// TIA Portal project "LavaCoches_IgnacioMorillasPadial_II" (V15)

(* hardware
DEVICE "S7300/ET200M station_1"  S7-300 station
   slot 0: "Perfil soporte_0"  Rail  6ES7 390-1***0-0AA0
   slot 2: "PLC_1"  CPU 314C-2 PN/DP  6ES7 314-6EH04-0AB0  V3.3
      slot 2: "Interfaz PROFINET_1"  PN-IO
         slot 1: "Port_1"  Port
         slot 2: "Port_2"  Port
      slot 5: "DI 24/DO 16_1"  DI24/DO16
      slot 6: "AI 5/AO 2_1"  AI5/AO2
      slot 7: "Contaje_1"  Counter
      slot 8: "Posicionamiento_1"  Positioning
*)

// ===== PLC "PLC_1"  CPU 314C-2 PN/DP =====

VAR_GLOBAL   // PLC tag table "STEP7 classic symbols"
   "CV2_FU" AT %I12.2 : Bool;   // Cepillo Vertical Izquierdo Fuera
   "CV2_Me" AT %I12.1 : Bool;   // Cepillo Vertical Izquierdo Medio
   "CV2_De" AT %I12.0 : Bool;   // Cepillo Vertical Izquierdo Dentro
   "V_Luz2" AT %I8.5 : Bool;   // Ventilador Sensor de Luz 2
   "V_Luz1" AT %I8.4 : Bool;   // Ventilador Sensor de Luz 1
   "CH_Abajo" AT %I8.3 : Bool;   // Cepillo Horizontal Sensor Magnético Abajo
   "CR2_Recoger" AT %Q9.3 : Bool;   // Cepillo Rueda Derecho Control Retirada
   "CR2_Salir" AT %Q9.2 : Bool;   // Ceplilo Rueda Derecho Control Salida
   "CR1_Recoger" AT %Q9.1 : Bool;   // Cepillo Rueda Izquierda Control Retirada
   "CV1_Fu" AT %I9.5 : Bool;   // Cepillo Vertical Derecho Fuera
   "CH_Bajar" AT %Q8.2 : Bool;   // Cepillo Horizontal Control Bajar
   "CRE_Avanzar" AT %Q8.1 : Bool;   // Cremallera Conrtol Avanzar
   "CRE_Retroceder" AT %Q8.0 : Bool;   // Cremallera Control Retroceder
   "CV2_R" AT %Q12.3 : Bool;   // Cepillo Vertical Derecho Rotar
   "CV1_De" AT %I9.7 : Bool;   // Cepillo Vertical Derecho Dentro
   "CV1_Me" AT %I9.6 : Bool;   // Cepillo Vertical Derecho Medio
   "CV2_Salir" AT %Q12.2 : Bool;   // Cepillo Vertical Izquierdo Salir
   "CR1_De" AT %I9.0 : Bool;   // Cepillo Rueda Derecha Dentro
   "V_Abajo" AT %I8.7 : Bool;   // Ventilador Sensor Magnético Abajo
   "V_Arriba" AT %I8.6 : Bool;   // Ventilador Sensor Magnético Arriba
   "Cont_CV" AT %MW10 : Int;   // Contador Ciclos CV
   "CV1_Salir" AT %Q12.1 : Bool;   // Cepillo Vertical Derecho Salir
   "CV1_R" AT %Q12.0 : Bool;   // Cepillo Vertical Derecho Rotar
   "CV1_Recoger" AT %Q9.7 : Bool;   // Cepillo Vertical Derecho Recoger
   "CH_Arriba" AT %I8.2 : Bool;   // Cepillo Horizontal Sensor Magnético Arriba
   "CH_Luz2" AT %I8.1 : Bool;   // Cepillo Horizontal Sensor de Luz 2
   "CH_Luz1" AT %I8.0 : Bool;   // Cepillo Horizontal Sensor de Luz 1
   "CR1_Salir" AT %Q9.0 : Bool;   // Cepillo Rueda Izquierda Control Salida
   "V_Subir" AT %Q8.7 : Bool;   // Ventilador Control Subir
   "CH_Subir" AT %Q8.6 : Bool;   // Cepillo Horizontal Control Subir
   "CV_Frente" AT %I12.7 : Bool;   // Cremallera Posción Labado Delante
   "CV_Atrás" AT %I12.6 : Bool;   // Cremallera Posción Labado Atrás
   "CR_Frente" AT %I12.5 : Bool;   // Cremallera Posición Ruedas Delanteras
   "CR2_Fu" AT %I9.2 : Bool;   // Cepillo Rueda Izquierda Fuera
   "CR2_De" AT %I9.3 : Bool;   // Cepillo Rueda Izquierda Dentro
   "CR1_Fu" AT %I9.1 : Bool;   // Cepillo Rueda Derecha Fuera
   "CH_R_+" AT %Q8.5 : Bool;   // Cepillo Horizontal Rotación Horaria
   "CH_R_-" AT %Q8.4 : Bool;   // Cepillo Horizontal Rotación Antihoraria
   "V_Bajar" AT %Q8.3 : Bool;   // Ventilador Control Bajar
   "CRE_Final" AT %I12.4 : Bool;   // Cremallera Posción Final
   "CRE_Inicio" AT %I12.3 : Bool;   // Cremallera Posición Inicio
   "CR_Atrás" AT %I13.0 : Bool;   // Cremallera Posción Ruedas Traseras
   "CV2_Recoger" AT %Q9.6 : Bool;   // Cepillo Vertical Izquierdo Recoger
   "CR2_R" AT %Q9.5 : Bool;   // Cepillo Izquierdo Rueda Rotación Horaria
   "CR1_R" AT %Q9.4 : Bool;   // Cepillo Derecho Rueda Rotación Horaria
   "CRE_Avanzar_CM" AT %M0.0 : Bool;
   "CRE_Retroceder_CM" AT %M0.2 : Bool;
   "CV1_Salir_CM" AT %M0.3 : Bool;
   "CV1_Recoger_CM" AT %M0.4 : Bool;
   "CV1_R_CM" AT %M0.5 : Bool;
   "CV2_Salir_CM" AT %M0.6 : Bool;
   "CV2_Recger_CM" AT %M0.7 : Bool;
   "CV2_R_CM" AT %M1.0 : Bool;
   "CH_Bajar_CM" AT %M1.1 : Bool;
   "CH_Subir_CM" AT %M1.2 : Bool;
   "CH_R_+_CM" AT %M1.3 : Bool;
   "CH_R_-_CM" AT %M1.4 : Bool;
   "V_Bajar_CM" AT %M1.5 : Bool;
   "V_Subir_CM" AT %M1.6 : Bool;
   "Reset_Maqueta" AT %M1.7 : Bool;
   "Automatico_Manual" AT %M0.1 : Bool;
   "AUX" AT %M2.0 : Bool;
   "AUX2" AT %M2.1 : Bool;
END_VAR

FUNCTION "Estructura horizontal" : Void   // FC1, SCL
{ S7_Optimized_Access := 'FALSE' }
VERSION : 0.1
BEGIN
   IF "CRE_Avanzar_CM" AND NOT "Automatico_Manual" THEN

       // sube hasta que ambos sensores opticos estan activos, o finalcarrera de arriba.
       IF "CH_Luz1" AND "CH_Luz2" THEN
           "CH_Subir_CM" := 0;
           "CH_Subir" := 0;
           "CH_Bajar_CM" := 1;
           "CH_Bajar" := 1;
       END_IF;

       // baja hasta que alguno de los sensores opticos mande una señal o llegue al final de carrera abajo.
       IF NOT "CH_Luz1" OR NOT "CH_Luz2" THEN
           "CH_Subir_CM" := 1;
           "CH_Subir" := 1;
       END_IF;
   END_IF;
   //Parada y recogidad de rodillo horizontal y activacion del ventilador
   //y finalizacion de FASE AVANCE y comienzo de RECOGIDA
   IF "CRE_Final" AND NOT "Automatico_Manual" THEN

       IF "CRE_Avanzar" AND "CRE_Avanzar_CM" THEN

           IF NOT "CH_Arriba" THEN
               "CH_R_+_CM" := 0;
               "CH_R_+" := 0;
               IF "CH_Bajar_CM" THEN
                   "CH_Bajar_CM" := 0;
                   "CH_Bajar" := 0;
               END_IF;

               IF NOT "CH_Subir_CM" THEN
                   "CH_Subir_CM" := 1;
                   "CH_Subir" := 1;
               END_IF;
           END_IF;
       END_IF;

       IF "CH_Arriba" THEN
           "CH_Subir_CM" := 0;
           "CH_Subir" := 0;
           "CRE_Retroceder_CM" := 1;
           "CRE_Retroceder" := 1;
           "V_Bajar_CM" := 1;
           "V_Bajar" := 1;
       END_IF;
   END_IF;

   IF "Reset_Maqueta" OR ("CRE_Inicio" AND NOT "Automatico_Manual") THEN
       "CH_R_+_CM" := 0;
       "CH_R_+" := 0;
       "CH_R_-_CM" := 0;
       "CH_R_-" := 0;
       IF NOT "CH_Arriba" THEN
           IF "CH_Bajar_CM" THEN
               "CH_Bajar_CM" := 0;
               "CH_Bajar" := 0;
           END_IF;
           "CH_Subir_CM" := 1;
           "CH_Subir" := 1;
       END_IF;

       IF "CH_Arriba" THEN
           "CH_Subir_CM" := 0;
           "CH_Subir" := 0;
           "CH_Bajar_CM" := 0;
           "CH_Bajar" := 0;
       END_IF;
   END_IF;

   IF NOT "AUX" AND "Automatico_Manual" THEN
       "CH_Subir_CM" := 0;
       "CH_Subir" := 0;
       "CH_Bajar_CM" := 0;
       "CH_Bajar" := 0;
   END_IF;


   //ACTIVACION DE ROTACION DE RODILLO HORIZONTAL
   //Comienza el giro y se activa la marca para que comience la actividad de subida y bajada
   IF ("CH_R_-_CM" AND NOT "CH_R_-") OR (NOT "CH_R_-_CM" AND "CH_R_-") THEN
       "CH_R_+_CM" := 0;
       "CH_R_+" := 0;
       "CH_R_-" := 1;
   END_IF;

   //Cambiar giro a horario
   IF ("CH_R_+_CM" AND NOT "CH_R_+") OR (NOT "CH_R_+_CM" AND "CH_R_+" ) THEN
       "CH_R_-_CM" := 0;
       "CH_R_-" := 0;
       "CH_R_+" := 1;
   END_IF;

   //para la bajada del Cepillo en e final de carrera
   IF ("CH_Bajar" OR "CH_Bajar_CM" ) AND ( NOT "CH_Luz1" OR NOT "CH_Luz2" OR "CH_Abajo" ) THEN
       "CH_Bajar_CM" := 0;
       "CH_Bajar" := 0;
   END_IF;

   //para la subida del ventilador en e final de carrera
   IF ("CH_Subir" OR "CH_Subir_CM") AND "CH_Arriba" THEN
       "CH_Subir_CM" := 0;
       "CH_Subir" := 0;
   END_IF;
END_FUNCTION

FUNCTION "Lavado vertical" : Void   // FC2, SCL
{ S7_Optimized_Access := 'FALSE' }
VERSION : 0.1
BEGIN
   IF "CRE_Avanzar_CM" AND NOT "Automatico_Manual"THEN

   /////////////////////////////////////////////////////
   //ENCARGADOS DE INICIAR LA ACCION
   ///////////////////////////////////////////////////////
   // Distingimos 2 casos:
   // - Parte delantera:
   //      Avanza el rodillo desde la posición mas afuera y comienza su rotacion
   IF "CV_Frente" AND "CV1_Fu" AND "CV2_FU" THEN

       //Rodillo 1
       "CV1_R_CM" := 1;
       "CV1_R" := 1;
       "CV1_Salir_CM" := 1;

       //Rodillo 2
       "CV2_R_CM" := 1;
       "CV2_R" := 1;
       "CV2_Salir_CM" := 1;

   END_IF;

   // - Parte trasera:
   //      Comienza su avance desde la posicion de medio (ya esta dando vueltas)
   IF "CV_Atrás" AND "Contador_repeticiones".CV = 3 THEN

       "CV1_Salir_CM" := 1;
       "CV2_Salir_CM" := 1;

   END_IF;

   /////////////////////////////////////////////////////
   //Movimiento hacia dentro de los RODILLOS VERICALES
   ///////////////////////////////////////////////////////
   IF "CV1_Salir_CM" AND ("CV1_Fu" OR "CV1_Me")THEN
       "CV1_Salir" := 1;
   END_IF;

   IF "CV2_Salir_CM" AND ("CV2_FU" OR "CV2_Me" ) THEN
       "CV2_Salir" := 1;
   END_IF;

   /////////////////////////////////////////////////////
   //Movimiento de recogida de RODILLOS VERICALES
   ///////////////////////////////////////////////////////

   IF NOT "CV2_Salir_CM" AND NOT "CV1_Salir_CM" AND "CV2_De" AND "CV1_De" THEN

       //Rodillo 1
       "CV1_Recoger_CM" := 1;
       "CV1_Recoger" := 1;

       //rodillo 2
       "CV2_Recger_CM" := 1;
       "CV2_Recoger" := 1;

   END_IF;

   /////////////////////////////////////////////////////
   //Parada de la accion recogida de RODILLOS VERICALES
   ///////////////////////////////////////////////////////

   //RODILLO 1
   // Dependiendo de las repeticiones, parará en la posicion fuera( en el caso del lavado trasero) o medio
   IF ("CV1_Recoger_CM" AND "CV1_Me" AND "Contador_repeticiones".CV >0) OR ("CV1_Recoger_CM" AND "CV1_Fu" AND "Contador_repeticiones".CV =0) THEN
       "CV1_Recoger_CM" := 0;
       "CV1_Recoger" := 0;

   END_IF;

   //RODILLO 2
   // Dependiendo de las repeticiones, parará en la posicion fuera( en el caso del lavado trasero esto pasará en su momento) o medio
   IF "CV2_Recger_CM" AND "CV2_Me" AND "Contador_repeticiones".CV >0 OR ("CV2_Recger_CM" AND "CV2_FU" AND "Contador_repeticiones".CV =0) THEN
       "CV2_Recger_CM" := 0;
       "CV2_Recoger" := 0;

   END_IF;

   /////////////////////////////////////////////////////
   //Condición de repeticion de RODILLOS VERICALES
   ///////////////////////////////////////////////////////

   //AMBOS CASOS (LAVADO FRONTAL Y TRASERO)
   //Mientras no haga 3 repeticiones estos volveran a contraerse
   IF ("CV1_Me" AND NOT "CV1_Recoger_CM" AND NOT "CV1_Salir_CM") AND ("CV2_Me" AND NOT "CV2_Recger_CM" AND NOT "CV2_Salir_CM") AND "Contador_repeticiones".CV>0 AND  "Contador_repeticiones".CV < 3 THEN
       "CV1_Salir_CM" := 1;
       "CV2_Salir_CM" := 1;
   END_IF;

   //CASO LAVADO FRONTAL
   //Cuando realice sus repeticiones la correa avanzrá y se le dala señal para que comience el cepillo horizontal
   IF ("CV1_Me" AND NOT "CV1_Recoger_CM" AND NOT "CV1_Salir_CM") AND ("CV2_Me" AND NOT "CV2_Recger_CM" AND NOT "CV2_Salir_CM") AND "Contador_repeticiones".CV >= 3 AND "CV_Frente" THEN
       "CRE_Avanzar" := 1;
       "CH_R_-_CM" := 1;
       "CH_Subir_CM" := 1;
   END_IF;

   //CASO LAVADO TRASERO
   //Cuando realice sus repeticiones la Correa avanzará, cambiaremos el giro del cepillo horizontal y
   //se para el giro de los cepillos verticales
   IF ("CV1_Fu" AND NOT "CV1_Recoger_CM" AND NOT "CV1_Salir_CM") AND ("CV2_FU" AND NOT "CV2_Recger_CM" AND NOT "CV2_Salir_CM") AND "Contador_repeticiones".CV = 0 AND "CV_Atrás" THEN
       "CRE_Avanzar" := 1;
       "CH_R_+_CM" := 1;
       "CV1_R_CM" := 0;
       "CV1_R" := 0;
       "CV2_R_CM" := 0;
       "CV2_R" := 0;
   END_IF;
   /////////////////////////////////////////////////////
   //CONTADOR DE REPETICIONES RODILLOS VERICALES
   ///////////////////////////////////////////////////////

   "Contador_repeticiones".CTUD(CU:="CV2_De" AND "CV1_De" AND "CV_Frente",
                                CD:="CV2_De" AND "CV1_De" AND "CV_Atrás",
                                R := ("CV1_Fu" AND "CV2_FU")OR "Reset_Maqueta",
                               PV:=3);

   END_IF;

   IF "Reset_Maqueta" THEN
       IF NOT "CV1_Fu" THEN
           "CV1_Salir_CM" := 0;
           "CV1_Salir" := 0;
           "CV1_Recoger_CM" := 1;
           "CV1_Recoger" := 1;
           "CV1_R_CM" := 0;
           "CV1_R" := 0;
       END_IF;
       IF "CV1_Fu" THEN
           "CV1_Recoger_CM" := 0;
           "CV1_Recoger" := 0;
           "CV1_Salir_CM" := 0;
           "CV1_Salir" := 0;
           "CV1_R_CM" := 0;
           "CV1_R" := 0;
       END_IF;

       IF NOT "CV2_FU" THEN
           "CV2_Salir_CM" := 0;
           "CV2_Salir" := 0;
           "CV2_Recger_CM" := 1;
           "CV2_Recoger" := 1;
           "CV2_R_CM" := 0;
           "CV2_R" := 0;
       END_IF;
       IF "CV2_FU" THEN
           "CV2_Recger_CM" := 0;
           "CV2_Recoger" := 0;
           "CV2_Salir_CM" := 0;
           "CV2_Salir" := 0;
           "CV2_R_CM" := 0;
           "CV2_R" := 0;
       END_IF;

   END_IF;

   IF NOT "AUX" AND "Automatico_Manual" THEN
       "CV2_Salir_CM" := 0;
       "CV2_Salir" := 0;
       "CV2_Recger_CM" := 0;
       "CV2_Recoger" := 0;

       "CV1_Recoger_CM" := 0;
       "CV1_Recoger" := 0;
       "CV1_Salir_CM" := 0;
       "CV1_Salir" := 0;
   END_IF;

   /////////////////////////////////////////////////////
   //Movimiento de parada al llegar Final de carrera de RODILLOS VERICALES
   ///////////////////////////////////////////////////////

   IF ("CV1_Salir_CM" OR "CV1_Salir") AND "CV1_De" OR ("CV1_Me" AND NOT ("CV_Frente" OR "CV_Atrás") )THEN
       "CV1_Salir_CM" := 0;
       "CV1_Salir" := 0;
   END_IF;

   IF (("CV2_Salir_CM" OR "CV2_Salir") AND "CV2_De") OR ("CV2_Me" AND NOT ("CV_Frente" OR "CV_Atrás")) THEN
       "CV2_Salir_CM" := 0;
       "CV2_Salir" := 0;
   END_IF;


   IF ("CV1_Recoger_CM" OR "CV1_Recoger") AND "CV1_Fu" THEN
       "CV1_Recoger_CM" := 0;
       "CV1_Recoger" := 0;
   END_IF;

   IF ("CV2_Recger_CM" OR "CV2_Recoger") AND "CV2_FU" THEN
       "CV2_Recger_CM" := 0;
       "CV2_Recoger" := 0;
   END_IF;
END_FUNCTION

FUNCTION "Lava_ruefas" : Void   // FC3, SCL
{ S7_Optimized_Access := 'FALSE' }
VERSION : 0.1
BEGIN
   IF "CRE_Avanzar_CM" AND NOT "Automatico_Manual" THEN

   //Salida de cepillo 1 y 2 con su giro, y frenado de cinta
   IF "CR1_De" AND "CR2_De" AND "CRE_Avanzar" AND (("contador_lava_rue".CV=0 AND "CR_Frente") OR ("contador_lava_rue".CV=1 AND "CR_Atrás") ) THEN
       "CRE_Avanzar" := 0;
       //rueda 1
       "CR1_Salir" := 1;
       "CR1_R" := 1;
       //rueda 2
       "CR2_Salir" := 1;
       "CR2_R" := 1;
   END_IF;

   //RECOGER DESPUES DE X TIEMPO
   //Cepillo 1
   IF "CR1_Fu" AND "T_1".Q THEN
       "CR1_Recoger" := 1;
       "CR1_R" := 0;
   END_IF;

   //Cepillo 2
   IF "CR2_Fu" AND "T_2".Q THEN
       // Statement section IF
       "CR2_Recoger" := 1;
       "CR2_R" := 0;
   END_IF;

   //continuar avanzando la cremayera
   IF "CR1_De" AND "CR2_De" AND NOT "CR1_Salir" AND NOT "CR2_Salir" AND NOT "CRE_Avanzar" AND (("contador_lava_rue".CV = 1 AND "CR_Frente") OR ("contador_lava_rue".CV = 0 AND "CR_Atrás")) THEN
       "CRE_Avanzar" := 1;

   END_IF;

   "contador_lava_rue".CTUD(CU:=("T_1" .Q OR "T_2".Q) AND "CR_Frente",
                            CD:=("T_1" .Q OR "T_2".Q) AND "CR_Atrás",
                            R:="Reset_Maqueta",
                            PV:=2);

   "T_1".TON(IN := "CR1_Fu",
             PT := T#1s);

   "T_2".TON(IN := "CR2_Fu",
             PT := T#1s);

   END_IF;

   IF "Reset_Maqueta" THEN
       "CR1_Salir" := 0;
       "CR2_Salir" := 0;
       "CR1_R" := 0;
       "CR2_R" := 0;
       //Recogida de ruedas
       IF NOT "CR1_De" THEN
           "CR1_Recoger" := 1;
       END_IF;

       IF NOT "CR2_De" THEN
           "CR2_Recoger" := 1;
       END_IF;
   END_IF;

   IF NOT "AUX" AND "Automatico_Manual" THEN
       "CR1_Salir" := 0;
       "CR2_Salir" := 0;
       "CR1_Recoger" := 0;
       "CR2_Recoger" := 0;
   END_IF;


   ////////////////////////////////////
   //DEJAR ESTADO FINAL
   //////////////////////////////////////
   IF "CR1_De" THEN
       "CR1_Recoger" := 0;
   END_IF;

   IF "CR2_De" THEN
       "CR2_Recoger" := 0;
   END_IF;

   ////////////////////////////////////
   //FRENADO DE FINAL DE CARRERA
   //////////////////////////////////////
   //Frenar final de carrera cepillo 1
   IF "CR1_Fu" THEN
       "CR1_Salir" := 0;
   END_IF;

   //Frenar final de carrera cepillo 2
   IF "CR2_Fu" THEN
       "CR2_Salir" := 0;
   END_IF;
END_FUNCTION

FUNCTION "ventiladorsecado" : Void   // FC4, SCL
{ S7_Optimized_Access := 'FALSE' }
VERSION : 0.1
BEGIN
   IF "CRE_Retroceder_CM" AND NOT "Automatico_Manual" THEN

       //Si los sensores opticos detectan, sube el ventilador
       //IF "CH_Luz1" AND "CH_Luz2" THEN
       IF NOT "V_Luz1" OR NOT "V_Luz2" THEN
           "V_Subir_CM" := 1;
           "V_Subir" :=1;
       END_IF;

       //Si los sensores no detectan baja elventilador
       IF "V_Luz1" AND  "V_Luz2" THEN
           // Statement section IF
           "V_Subir_CM" := 0;
           "V_Subir" := 0;
           "V_Bajar_CM" := 1;
           "V_Bajar" := 1;
       END_IF;

   END_IF;

   IF "CRE_Inicio" OR "Reset_Maqueta" THEN
       //"CRE_Retroceder_CM" := 0;
       //"CRE_Retroceder" := 0;
       "V_Bajar" := 0;
       "V_Bajar_CM" := 0;

       IF NOT "V_Arriba" THEN
           "V_Subir_CM" := 1;
           "V_Subir" := 1;
       END_IF;

   END_IF;

   IF NOT "AUX" AND "Automatico_Manual" THEN
       "V_Bajar" := 0;
       "V_Bajar_CM" := 0;
       "V_Subir_CM" := 0;
       "V_Subir" := 0;
   END_IF;

   //para la bajada del ventilador en e final de carrera
   IF ("V_Bajar" OR "V_Bajar_CM") AND (NOT "V_Luz1" OR NOT "V_Luz2" OR  "V_Abajo") THEN
       "V_Bajar_CM" := 0;
       "V_Bajar" := 0;
   END_IF;

   IF "V_Arriba" THEN
       "V_Subir_CM" := 0;
       "V_Subir" := 0;
   END_IF;
END_FUNCTION

FUNCTION "tratamiento" : Void   // FC5, SCL
{ S7_Optimized_Access := 'FALSE' }
VERSION : 0.1
BEGIN
   "Estructura horizontal"();
   "Lava_ruefas"();
   "Lavado vertical"();
   "ventiladorsecado"();
   IF  NOT "Automatico_Manual" OR (NOT "AUX" AND "Automatico_Manual") THEN
       "CRE_Retroceder_CM" := 0;
       "CRE_Retroceder" := 0;
       "CRE_Avanzar_CM" := 0;
       "CRE_Avanzar" := 0;
   END_IF;
END_FUNCTION

ORGANIZATION_BLOCK "Main"   // OB1, SCL
TITLE = "Main Program Sweep (Cycle)"
{ S7_Optimized_Access := 'FALSE' }
VERSION : 0.1
   VAR_TEMP
      OB1_EV_CLASS : Byte;   // Bits 0-3 = 1 (Coming event), Bits 4-7 = 1 (Event class 1)
      OB1_SCAN_1 : Byte;   // 1 (Cold restart scan 1 of OB 1), 3 (Scan 2-n of OB 1)
      OB1_PRIORITY : Byte;   // Priority of OB Execution
      OB1_OB_NUMBR : Byte;   // 1 (Organization block 1, OB1)
      OB1_RESERVED_1 : Byte;   // Reserved for system
      OB1_RESERVED_2 : Byte;   // Reserved for system
      OB1_PREV_CYCLE : Int;   // Cycle time of previous OB1 scan (milliseconds)
      OB1_MIN_CYCLE : Int;   // Minimum cycle time of OB1 (milliseconds)
      OB1_MAX_CYCLE : Int;   // Maximum cycle time of OB1 (milliseconds)
      OB1_DATE_TIME : Date_And_Time;   // Date and time OB1 started
   END_VAR
BEGIN
   //Establece la situacion inicial, poniendo las marcas existentes a false y el arranque de la cremayera.
   //Tambien se encarga de restablecer la posición del retocreso de la maqueta.
   //NOTA: Entre otras cosas,esto lo hago para no tener que estar desactivando a mano las señales en el PLC cuando hago un reset,Ya que
   //si funciona correctamente solo estará activado la que funcione en ese instante, por lo que no sería necesario.

   IF NOT "Automatico_Manual" THEN
       IF "AUX" THEN
           "AUX" := 0;
           "Reset_Maqueta" := 1;
       END_IF;


   IF "CRE_Inicio" THEN
       IF "Reset_Maqueta" AND ("CRE_Retroceder" OR "CRE_Retroceder_CM") THEN
           "CRE_Retroceder" := 0;
           "CRE_Retroceder_CM" := 0;
       END_IF;

       IF NOT ("CV1_Fu" AND "CV2_FU" AND "CH_Arriba" AND "V_Arriba" AND "CR2_De" AND "CR1_De") THEN
           "Reset_Maqueta" := 1;
           "tratamiento"();
       ELSE
           "tratamiento"();
           "Reset_Maqueta" := 0;
           "CRE_Avanzar_CM" := 1;
           "CRE_Avanzar" := 1;
       END_IF;


   END_IF;

   //Este apartado engloba todo lo correspondiente con las actividades de avance
   IF "CRE_Avanzar_CM" AND NOT "CRE_Inicio" THEN

       // Se para y activa el lavado de los rodillos verticales.
       IF "CV_Frente" THEN
           "CRE_Avanzar" := 0;
           "Lavado vertical"();
       END_IF;

       //Se encarga de regular la altura del cepillo horizontal
       IF "CH_R_-_CM" OR "CH_R_+_CM" THEN
           "Estructura horizontal"();
       END_IF;

       //Lavado de ruedas delanteras
       //Frena el avance de cremallera
       IF "CR_Frente" THEN
           "Lava_ruefas"();
       END_IF;

       //Lavado trasero y parada
       IF "CV_Atrás" THEN
           "CRE_Avanzar" := 0;
           "Lavado vertical"();
       END_IF;

       //Lavado ruedas atras
       IF "CR_Atrás" THEN
           "Lava_ruefas"();
       END_IF;

   END_IF;

   IF "CRE_Final" THEN
       "CRE_Avanzar_CM" := 0;
       "CRE_Avanzar" := 0;
       "Estructura horizontal"();
   END_IF;


   IF "CRE_Retroceder_CM" THEN
       "ventiladorsecado"();
   END_IF;

   END_IF;

   IF "Automatico_Manual" THEN
       "tratamiento"();
       "AUX" := 1;
   END_IF;

   IF "Reset_Maqueta" THEN
       IF NOT ("CV1_Fu" AND "CV2_FU" AND "CH_Arriba" AND "V_Arriba" AND "CR2_De" AND "CR1_De") THEN
           "tratamiento"();
           //  "Reset_Maqueta" := 1;
       ELSE
           "tratamiento"();
           "CRE_Retroceder" := 1;
           IF "CRE_Inicio" THEN
               "Reset_Maqueta" := 0;
           END_IF;



       END_IF;
   END_IF;


   IF "CRE_Final" THEN
       "CRE_Avanzar_CM" := 0;
       "CRE_Avanzar" := 0;
   END_IF;

   IF "CRE_Inicio" THEN
       "CRE_Retroceder_CM" := 0;
       "CRE_Retroceder" := 0;
   END_IF;
END_ORGANIZATION_BLOCK